SUBAPPLICATION Uebung_002c (* DigitalInput_I1/_I2 auf DigitalOutput_Q1 *)
  (* Standard: 61499-2 *)
  (* Version 1.0, 2023-10-23, franz *)
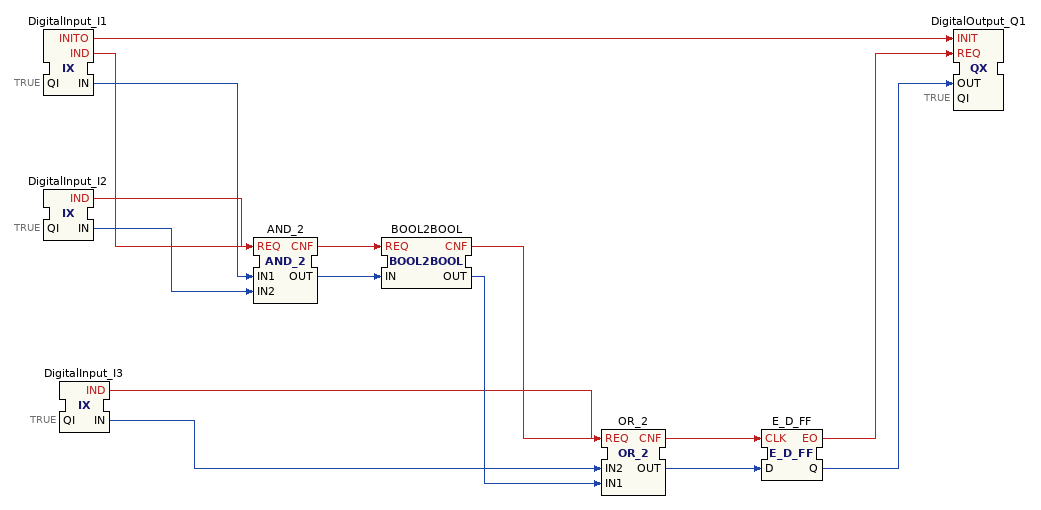
  FBS
    DigitalOutput_Q1 : QX(QI := TRUE);
    DigitalInput_I1 : IX(QI := TRUE);
    DigitalInput_I2 : IX(QI := TRUE);
    AND_2 : AND_2;
    DigitalInput_I3 : IX(QI := TRUE);
    OR_2 : OR_2;
    BOOL2BOOL : BOOL2BOOL;
    E_D_FF : E_D_FF;
  END_FBS
  EVENT_CONNECTIONS
    DigitalInput_I1.INITO TO DigitalOutput_Q1.INIT;
    DigitalInput_I1.IND TO AND_2.REQ;
    DigitalInput_I2.IND TO AND_2.REQ;
    E_D_FF.EO TO DigitalOutput_Q1.REQ;
    AND_2.CNF TO BOOL2BOOL.REQ;
    BOOL2BOOL.CNF TO OR_2.REQ;
    DigitalInput_I3.IND TO OR_2.REQ;
    OR_2.CNF TO E_D_FF.CLK;
  END_CONNECTIONS
  DATA_CONNECTIONS
    DigitalInput_I1.IN TO AND_2.IN1;
    DigitalInput_I2.IN TO AND_2.IN2;
    DigitalInput_I3.IN TO OR_2.IN2;
    E_D_FF.Q TO DigitalOutput_Q1.OUT;
    AND_2.OUT TO BOOL2BOOL.IN;
    BOOL2BOOL.OUT TO OR_2.IN1;
    OR_2.OUT TO E_D_FF.D;
  END_CONNECTIONS
END_SUBAPPLICATION
